FUNCTION_BLOCK INTERNAL FB_SL3K4_Test EXTENDS FB_TestSuite
VAR
    testStage1    : ST_MCS2Stage;
    testStage2    : ST_MCS2Stage;
    testStage3    : ST_MCS2Stage;
    testStage4    : ST_MCS2Stage;
	testStage5    : REFERENCE TO ST_MotionStage;
    fbFFHWO       : FB_HardwareFFOutput;
    fbArbiter     : FB_Arbiter(1);
    astDummyBeam  : ARRAY[0..2] OF ST_DbStateParams;
    fbTestHelper  : FB_PMPSJsonTestHelper;
    fbSubSysIO    : FB_DummyArbIO;
    testFB        : FB_SL3K4;
    n         : INT;
    driftAxis : INT;
	
    devName        : STRING := 'SL3K4';
	fbReadTimer : TON := (PT:=T#1S);
	fbTestTimer: TON := (IN:=TRUE, PT:=T#4S);
	nTestStep : UINT;
	
END_VAR

TEST(__POUNAME());
	// Prepare dummy beam parameter sets
	astDummyBeam[E_SL3K4State.NORMAL].stBeamParams.nBCRange         := 16#7FFF;    // All 15 classes
	astDummyBeam[E_SL3K4State.NORMAL].stBeamParams.nTran            := 15;
	astDummyBeam[E_SL3K4State.NORMAL].stBeamParams.nRate            := 120;
	astDummyBeam[E_SL3K4State.NORMAL].nRequestAssertionID           := 2;
	astDummyBeam[E_SL3K4State.NORMAL].sPmpsState                    := 'NORMAL';
	
	astDummyBeam[E_SL3K4State.MAINTENANCE].stBeamParams.nBCRange    := 16#0040;    // Only class 6
	astDummyBeam[E_SL3K4State.MAINTENANCE].stBeamParams.nTran       := 0.01;
	astDummyBeam[E_SL3K4State.MAINTENANCE].stBeamParams.nRate       := 0;
	astDummyBeam[E_SL3K4State.MAINTENANCE].nRequestAssertionID      := 3;
	astDummyBeam[E_SL3K4State.MAINTENANCE].sPmpsState               := 'MAINTENANCE';

	astDummyBeam[E_SL3K4State.TRANSITION].nRequestAssertionID       := 1;
	astDummyBeam[E_SL3K4State.TRANSITION].stBeamParams              := PMPS_GVL.cst0RateBeam;
	astDummyBeam[E_SL3K4State.TRANSITION].sPmpsState                := 'TRANSITION';
	fbTestHelper.sDevName := 'SL3K4';

//testStage5 REF= testStage1;
CASE nTestStep OF
	0:
		// Write dummy beam assertions to test location
		fbTestHelper.bExecute := TRUE;
		testFB.bFileReaderBusy := TRUE;
		nTestStep := 1;
	1:
		fbReadTimer.IN:=TRUE;
		nTestStep := 2;
	2:
		IF 	fbReadTimer.Q THEN
			testFB.bFileReaderBusy := FALSE;
			fbTestHelper.bExecute := FALSE;
			nTestStep := 3;
		END_IF
	
END_CASE

fbReadTimer();
fbTestHelper(
	astBeamParams := astDummyBeam,
);

testFB(
   stX1    := testStage1,
   stX2 := testStage2,
   stY1  := testStage3,
   stY2  := testStage4,
   bFileReaderError := FALSE,
   sTransitionKey   := 'TRANSITION',
   fbFFHWO       := fbFFHWO,
   fbArbiter     := fbArbiter,
);

fbSubSysIO(LA := fbArbiter, FFO := fbFFHWO);
 
IF fbTestTimer.Q THEN

    TEST_FINISHED();
END_IF

END_FUNCTION_BLOCK

(* stored: Version 1.1.0.1
   POU FB_SL3K4_Test: Id {4cd567df-faf8-4c92-a022-7ee8ed605221}, SpecialFunc None *)
